FUNCTION_BLOCK FB_TempSensPt100 IMPLEMENTS I_TemperatureSensor
VAR_INPUT
	TempRaw AT %I* : REAL;
END_VAR
VAR_OUTPUT
END_VAR
VAR
	//Properties
	fTemperature : REAL;
	//Raw value
	
END_VAR

METHOD Run
//Read temperature
fTemperature :=  FC_Pt100Raw_TO_Temperature(TempRaw);
END_METHOD

PROPERTY Temperature : REAL
GET
Temperature := THIS^.fTemperature;
END_GET
SET
END_SET
END_PROPERTY

END_FUNCTION_BLOCK

(* stored: Version 1.1.0.1, ProductVersion 3.1.4024.3
   POU FB_TempSensPt100: Id {1270eee1-cc09-4dcf-b2ee-a46bbf247da3}, SpecialFunc None
   Method Run: Id {69f66fdc-0e32-4839-b055-1133c20a82d5}
   Property Temperature: Id {4a7ad6b5-bc3c-4562-896a-e62a1a07b1bb}
   Get Get: Id {9229b9c9-be72-4301-9602-0cf196997142}
   Set Set: Id {f5065692-367a-4616-a02c-46d13d8eab2a} *)
